TYPE C2000_ANALOG_OUTPUTS :
STRUCT
	
	AFM : REAL;

END_STRUCT
END_TYPE

(* stored: Version 1.1.0.1, ProductVersion 3.1.4024.15
   DUT C2000_ANALOG_OUTPUTS: Id {df94ce26-80a1-0b69-374a-5290d50b6a7d} *)
